// TIA Portal V17 export
// export: Created 2023-10-17T06:55:20.3967986Z, ExportSetting WithDefaults, DisplayName Totally Integrated Automation Portal, DisplayVersion V17, DisplayName TIA Portal Openness, DisplayVersion V17, DisplayName TIA Portal Version Control Interface, DisplayVersion V17, DisplayName STEP 7 Professional, DisplayVersion V17, DisplayName STEP 7 Safety, DisplayVersion V17, DisplayName WinCC Advanced, DisplayVersion V17
ORGANIZATION_BLOCK "Main"   // OB1, LAD, ProgramCycle
TITLE = "Main Program Sweep (Cycle)"
{ S7_Optimized_Access := 'TRUE' }
VERSION : 0.1
// stored: AutoNumber true, IsIECCheckEnabled false, SetENOAutomatically false
   VAR_INPUT
      Initial_Call : Bool;   // Initial call of this OB
      Remanence : Bool;   // =True, if remanent data are available
   END_VAR
   VAR_TEMP
      "Auto/Manual" : Bool;
   END_VAR
   VAR_TEMP   // added for the SCL form of the ladder/FBD networks
      _w1 : Bool;
   END_VAR
BEGIN

REGION Network 1
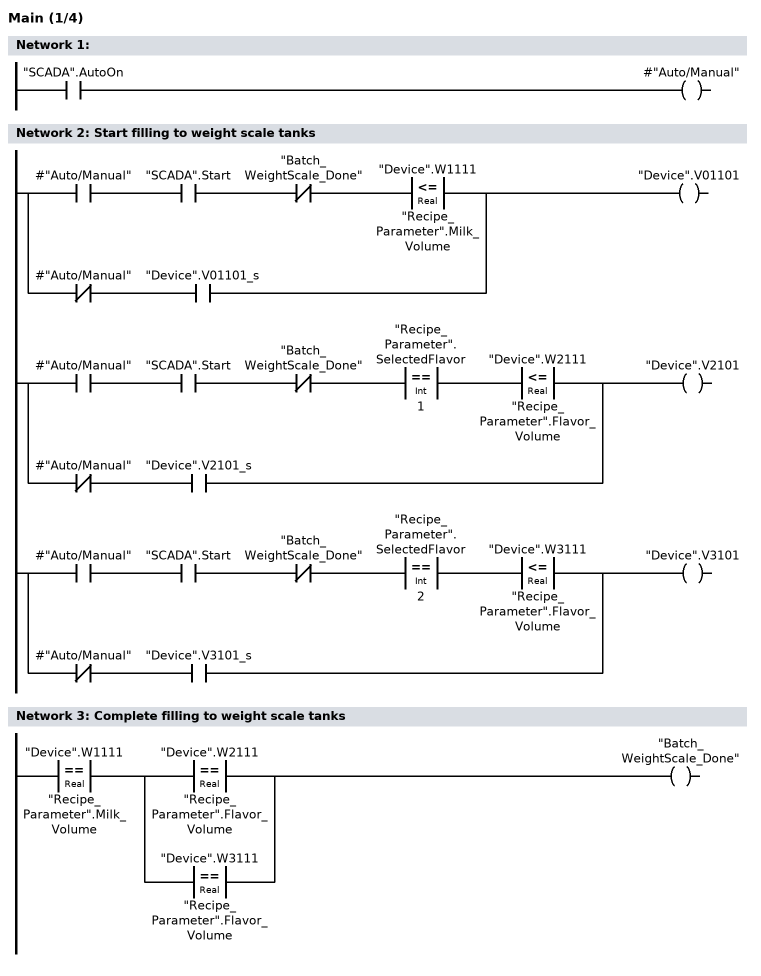
   RUNG wire#powerrail
      Contact( "SCADA".AutoOn )
      Coil( #"Auto/Manual" )
   END_RUNG
   // the same network as SCL:
   #"Auto/Manual" := "SCADA".AutoOn;
END_REGION

REGION Network 2: Start filling to weight scale tanks
   RUNG wire#powerrail
      Contact( #"Auto/Manual" )
      Contact( "SCADA".Start )
      I_Contact( "Batch_WeightScale_Done" )
      { S7_Templates := "SrcType := Real" } LE_Contact(in1 := "Device".W1111, in2 := "Recipe_Parameter".Milk_Volume)
      wire#w1
      Coil( "Device".V01101 )
   END_RUNG
   RUNG wire#powerrail
      I_Contact( #"Auto/Manual" )
      Contact( "Device".V01101_s )
   END_RUNG wire#w1
   RUNG wire#powerrail
      Contact( #"Auto/Manual" )
      Contact( "SCADA".Start )
      I_Contact( "Batch_WeightScale_Done" )
      { S7_Templates := "SrcType := Int" } EQ_Contact(in1 := "Recipe_Parameter".SelectedFlavor, in2 := 1)
      { S7_Templates := "SrcType := Real" } LE_Contact(in1 := "Device".W2111, in2 := "Recipe_Parameter".Flavor_Volume)
      wire#w2
      Coil( "Device".V2101 )
   END_RUNG
   RUNG wire#powerrail
      I_Contact( #"Auto/Manual" )
      Contact( "Device".V2101_s )
   END_RUNG wire#w2
   RUNG wire#powerrail
      Contact( #"Auto/Manual" )
      Contact( "SCADA".Start )
      I_Contact( "Batch_WeightScale_Done" )
      { S7_Templates := "SrcType := Int" } EQ_Contact(in1 := "Recipe_Parameter".SelectedFlavor, in2 := 2)
      { S7_Templates := "SrcType := Real" } LE_Contact(in1 := "Device".W3111, in2 := "Recipe_Parameter".Flavor_Volume)
      wire#w3
      Coil( "Device".V3101 )
   END_RUNG
   RUNG wire#powerrail
      I_Contact( #"Auto/Manual" )
      Contact( "Device".V3101_s )
   END_RUNG wire#w3
   // the same network as SCL:
   "Device".V01101 := (#"Auto/Manual" AND "SCADA".Start AND NOT "Batch_WeightScale_Done" AND ("Device".W1111 <= "Recipe_Parameter".Milk_Volume)) OR (NOT #"Auto/Manual" AND "Device".V01101_s);
   "Device".V2101 := (#"Auto/Manual" AND "SCADA".Start AND NOT "Batch_WeightScale_Done" AND ("Recipe_Parameter".SelectedFlavor = 1) AND ("Device".W2111 <= "Recipe_Parameter".Flavor_Volume)) OR (NOT #"Auto/Manual" AND "Device".V2101_s);
   "Device".V3101 := (#"Auto/Manual" AND "SCADA".Start AND NOT "Batch_WeightScale_Done" AND ("Recipe_Parameter".SelectedFlavor = 2) AND ("Device".W3111 <= "Recipe_Parameter".Flavor_Volume)) OR (NOT #"Auto/Manual" AND "Device".V3101_s);
END_REGION

REGION Network 3: Complete filling to weight scale tanks
   RUNG wire#powerrail
      { S7_Templates := "SrcType := Real" } EQ_Contact(in1 := "Device".W1111, in2 := "Recipe_Parameter".Milk_Volume)
      wire#w1
      { S7_Templates := "SrcType := Real" } EQ_Contact(in1 := "Device".W2111, in2 := "Recipe_Parameter".Flavor_Volume)
      wire#w2
      Coil( "Batch_WeightScale_Done" )
   END_RUNG
   RUNG wire#w1
      { S7_Templates := "SrcType := Real" } EQ_Contact(in1 := "Device".W3111, in2 := "Recipe_Parameter".Flavor_Volume)
   END_RUNG wire#w2
   // the same network as SCL:
   "Batch_WeightScale_Done" := ("Device".W1111 = "Recipe_Parameter".Milk_Volume) AND (("Device".W2111 = "Recipe_Parameter".Flavor_Volume) OR ("Device".W3111 = "Recipe_Parameter".Flavor_Volume));
END_REGION

REGION Network 4: Start filling the mixer
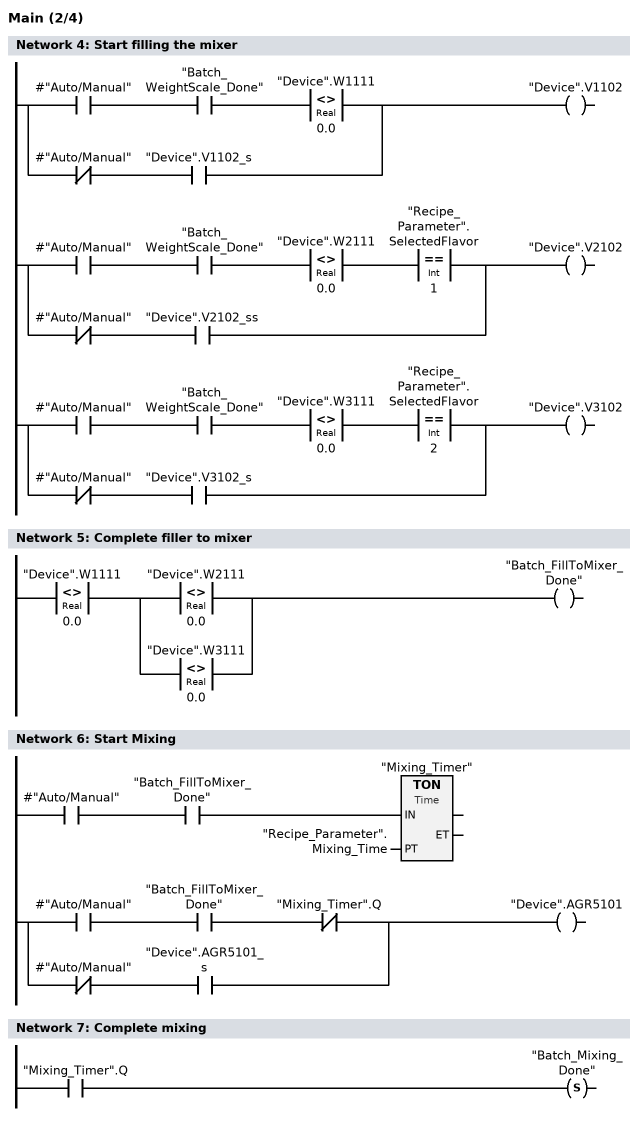
   RUNG wire#powerrail
      Contact( #"Auto/Manual" )
      Contact( "Batch_WeightScale_Done" )
      { S7_Templates := "SrcType := Real" } NE_Contact(in1 := "Device".W1111, in2 := 0.0)
      wire#w1
      Coil( "Device".V1102 )
   END_RUNG
   RUNG wire#powerrail
      I_Contact( #"Auto/Manual" )
      Contact( "Device".V1102_s )
   END_RUNG wire#w1
   RUNG wire#powerrail
      Contact( #"Auto/Manual" )
      Contact( "Batch_WeightScale_Done" )
      { S7_Templates := "SrcType := Real" } NE_Contact(in1 := "Device".W2111, in2 := 0.0)
      { S7_Templates := "SrcType := Int" } EQ_Contact(in1 := "Recipe_Parameter".SelectedFlavor, in2 := 1)
      wire#w2
      Coil( "Device".V2102 )
   END_RUNG
   RUNG wire#powerrail
      I_Contact( #"Auto/Manual" )
      Contact( "Device".V2102_ss )
   END_RUNG wire#w2
   RUNG wire#powerrail
      Contact( #"Auto/Manual" )
      Contact( "Batch_WeightScale_Done" )
      { S7_Templates := "SrcType := Real" } NE_Contact(in1 := "Device".W3111, in2 := 0.0)
      { S7_Templates := "SrcType := Int" } EQ_Contact(in1 := "Recipe_Parameter".SelectedFlavor, in2 := 2)
      wire#w3
      Coil( "Device".V3102 )
   END_RUNG
   RUNG wire#powerrail
      I_Contact( #"Auto/Manual" )
      Contact( "Device".V3102_s )
   END_RUNG wire#w3
   // the same network as SCL:
   "Device".V1102 := (#"Auto/Manual" AND "Batch_WeightScale_Done" AND ("Device".W1111 <> 0.0)) OR (NOT #"Auto/Manual" AND "Device".V1102_s);
   "Device".V2102 := (#"Auto/Manual" AND "Batch_WeightScale_Done" AND ("Device".W2111 <> 0.0) AND ("Recipe_Parameter".SelectedFlavor = 1)) OR (NOT #"Auto/Manual" AND "Device".V2102_ss);
   "Device".V3102 := (#"Auto/Manual" AND "Batch_WeightScale_Done" AND ("Device".W3111 <> 0.0) AND ("Recipe_Parameter".SelectedFlavor = 2)) OR (NOT #"Auto/Manual" AND "Device".V3102_s);
END_REGION

REGION Network 5: Complete filler to mixer
   RUNG wire#powerrail
      { S7_Templates := "SrcType := Real" } NE_Contact(in1 := "Device".W1111, in2 := 0.0)
      wire#w1
      { S7_Templates := "SrcType := Real" } NE_Contact(in1 := "Device".W2111, in2 := 0.0)
      wire#w2
      Coil( "Batch_FillToMixer_Done" )
   END_RUNG
   RUNG wire#w1
      { S7_Templates := "SrcType := Real" } NE_Contact(in1 := "Device".W3111, in2 := 0.0)
   END_RUNG wire#w2
   // the same network as SCL:
   "Batch_FillToMixer_Done" := ("Device".W1111 <> 0.0) AND (("Device".W2111 <> 0.0) OR ("Device".W3111 <> 0.0));
END_REGION

REGION Network 6: Start Mixing
   RUNG wire#powerrail
      Contact( #"Auto/Manual" )
      Contact( "Batch_FillToMixer_Done" )
      { S7_Templates := "time_type := Time" } "Mixing_Timer".TON(pt := "Recipe_Parameter".Mixing_Time, et =>)
   END_RUNG
   RUNG wire#powerrail
      Contact( #"Auto/Manual" )
      Contact( "Batch_FillToMixer_Done" )
      I_Contact( "Mixing_Timer".Q )
      wire#w1
      Coil( "Device".AGR5101 )
   END_RUNG
   RUNG wire#powerrail
      I_Contact( #"Auto/Manual" )
      Contact( "Device".AGR5101_s )
   END_RUNG wire#w1
   // the same network as SCL:
   "Mixing_Timer".TON(IN := #"Auto/Manual" AND "Batch_FillToMixer_Done", PT := "Recipe_Parameter".Mixing_Time);
   "Device".AGR5101 := (#"Auto/Manual" AND "Batch_FillToMixer_Done" AND NOT "Mixing_Timer".Q) OR (NOT #"Auto/Manual" AND "Device".AGR5101_s);
END_REGION

REGION Network 7: Complete mixing
   RUNG wire#powerrail
      Contact( "Mixing_Timer".Q )
      S_Coil( "Batch_Mixing_Done" )
   END_RUNG
   // the same network as SCL:
   IF "Mixing_Timer".Q THEN "Batch_Mixing_Done" := TRUE; END_IF;
END_REGION

REGION Network 8: Start filling to pasteurising machine
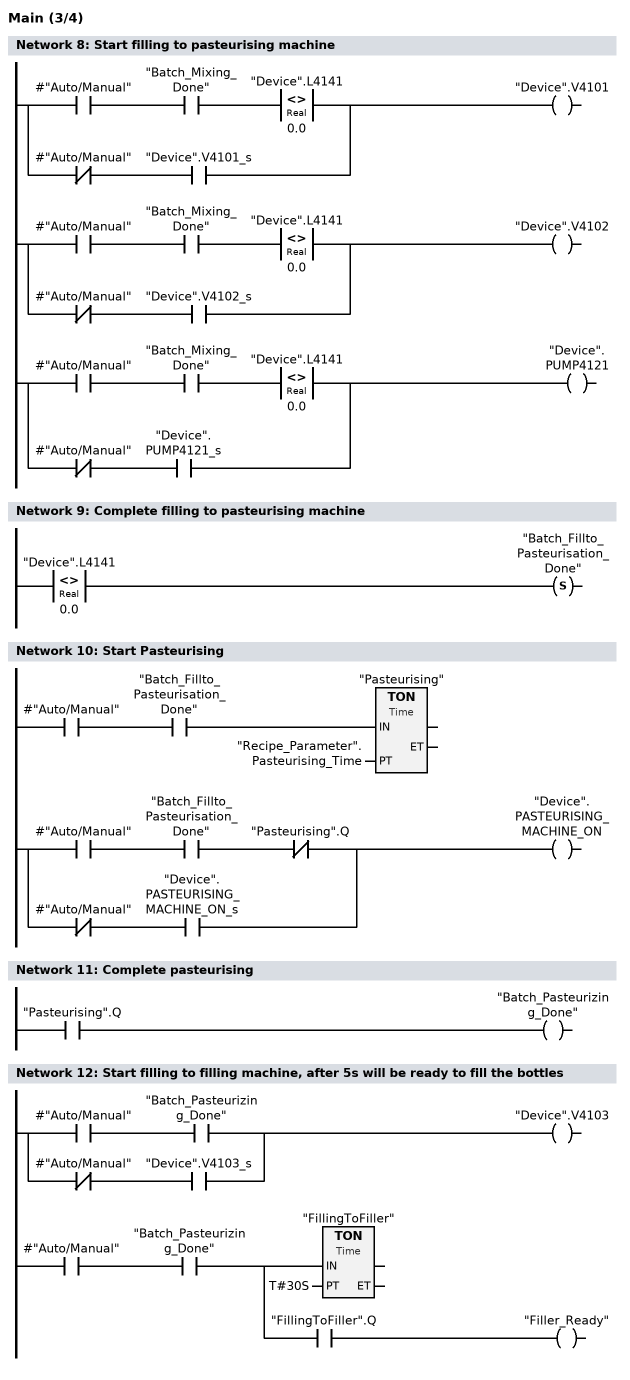
   RUNG wire#powerrail
      Contact( #"Auto/Manual" )
      Contact( "Batch_Mixing_Done" )
      { S7_Templates := "SrcType := Real" } NE_Contact(in1 := "Device".L4141, in2 := 0.0)
      wire#w1
      Coil( "Device".V4101 )
   END_RUNG
   RUNG wire#powerrail
      I_Contact( #"Auto/Manual" )
      Contact( "Device".V4101_s )
   END_RUNG wire#w1
   RUNG wire#powerrail
      Contact( #"Auto/Manual" )
      Contact( "Batch_Mixing_Done" )
      { S7_Templates := "SrcType := Real" } NE_Contact(in1 := "Device".L4141, in2 := 0.0)
      wire#w2
      Coil( "Device".V4102 )
   END_RUNG
   RUNG wire#powerrail
      I_Contact( #"Auto/Manual" )
      Contact( "Device".V4102_s )
   END_RUNG wire#w2
   RUNG wire#powerrail
      Contact( #"Auto/Manual" )
      Contact( "Batch_Mixing_Done" )
      { S7_Templates := "SrcType := Real" } NE_Contact(in1 := "Device".L4141, in2 := 0.0)
      wire#w3
      Coil( "Device".PUMP4121 )
   END_RUNG
   RUNG wire#powerrail
      I_Contact( #"Auto/Manual" )
      Contact( "Device".PUMP4121_s )
   END_RUNG wire#w3
   // the same network as SCL:
   "Device".V4101 := (#"Auto/Manual" AND "Batch_Mixing_Done" AND ("Device".L4141 <> 0.0)) OR (NOT #"Auto/Manual" AND "Device".V4101_s);
   "Device".V4102 := (#"Auto/Manual" AND "Batch_Mixing_Done" AND ("Device".L4141 <> 0.0)) OR (NOT #"Auto/Manual" AND "Device".V4102_s);
   "Device".PUMP4121 := (#"Auto/Manual" AND "Batch_Mixing_Done" AND ("Device".L4141 <> 0.0)) OR (NOT #"Auto/Manual" AND "Device".PUMP4121_s);
END_REGION

REGION Network 9: Complete filling to pasteurising machine
   RUNG wire#powerrail
      { S7_Templates := "SrcType := Real" } NE_Contact(in1 := "Device".L4141, in2 := 0.0)
      S_Coil( "Batch_Fillto_Pasteurisation_Done" )
   END_RUNG
   // the same network as SCL:
   IF "Device".L4141 <> 0.0 THEN "Batch_Fillto_Pasteurisation_Done" := TRUE; END_IF;
END_REGION

REGION Network 10: Start Pasteurising
   RUNG wire#powerrail
      Contact( #"Auto/Manual" )
      Contact( "Batch_Fillto_Pasteurisation_Done" )
      { S7_Templates := "time_type := Time" } "Pasteurising".TON(pt := "Recipe_Parameter".Pasteurising_Time, et =>)
   END_RUNG
   RUNG wire#powerrail
      Contact( #"Auto/Manual" )
      Contact( "Batch_Fillto_Pasteurisation_Done" )
      I_Contact( "Pasteurising".Q )
      wire#w1
      Coil( "Device".PASTEURISING_MACHINE_ON )
   END_RUNG
   RUNG wire#powerrail
      I_Contact( #"Auto/Manual" )
      Contact( "Device".PASTEURISING_MACHINE_ON_s )
   END_RUNG wire#w1
   // the same network as SCL:
   "Pasteurising".TON(IN := #"Auto/Manual" AND "Batch_Fillto_Pasteurisation_Done",
                      PT := "Recipe_Parameter".Pasteurising_Time);
   "Device".PASTEURISING_MACHINE_ON := (#"Auto/Manual" AND "Batch_Fillto_Pasteurisation_Done" AND NOT "Pasteurising".Q) OR (NOT #"Auto/Manual" AND "Device".PASTEURISING_MACHINE_ON_s);
END_REGION

REGION Network 11: Complete pasteurising
   RUNG wire#powerrail
      Contact( "Pasteurising".Q )
      Coil( "Batch_Pasteurizing_Done" )
   END_RUNG
   // the same network as SCL:
   "Batch_Pasteurizing_Done" := "Pasteurising".Q;
END_REGION

REGION Network 12: Start filling to filling machine, after 5s will be ready to fill the bottles
   RUNG wire#powerrail
      Contact( #"Auto/Manual" )
      Contact( "Batch_Pasteurizing_Done" )
      wire#w1
      Coil( "Device".V4103 )
   END_RUNG
   RUNG wire#powerrail
      I_Contact( #"Auto/Manual" )
      Contact( "Device".V4103_s )
   END_RUNG wire#w1
   RUNG wire#powerrail
      Contact( #"Auto/Manual" )
      Contact( "Batch_Pasteurizing_Done" )
      wire#w2
      { S7_Templates := "time_type := Time" } "FillingToFiller".TON(pt := T#30S, et =>)
   END_RUNG
   RUNG wire#w2
      Contact( "FillingToFiller".Q )
      Coil( "Filler_Ready" )
   END_RUNG
   // the same network as SCL:
   "Device".V4103 := (#"Auto/Manual" AND "Batch_Pasteurizing_Done") OR (NOT #"Auto/Manual" AND "Device".V4103_s);
   #_w1 := #"Auto/Manual" AND "Batch_Pasteurizing_Done";
   "FillingToFiller".TON(IN := #_w1, PT := T#30S);
   "Filler_Ready" := #_w1 AND "FillingToFiller".Q;
END_REGION

REGION Network 13: Run filler until level of feed until 0.5 liters
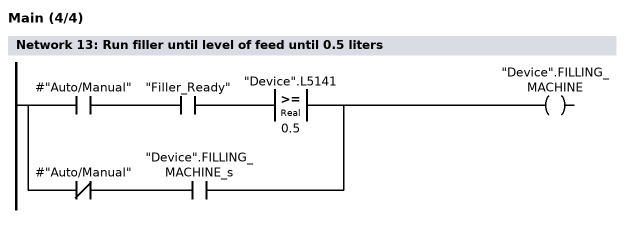
   RUNG wire#powerrail
      Contact( #"Auto/Manual" )
      Contact( "Filler_Ready" )
      { S7_Templates := "SrcType := Real" } GE_Contact(in1 := "Device".L5141, in2 := 0.5)
      wire#w1
      Coil( "Device".FILLING_MACHINE )
   END_RUNG
   RUNG wire#powerrail
      I_Contact( #"Auto/Manual" )
      Contact( "Device".FILLING_MACHINE_s )
   END_RUNG wire#w1
   // the same network as SCL:
   "Device".FILLING_MACHINE := (#"Auto/Manual" AND "Filler_Ready" AND ("Device".L5141 >= 0.5)) OR (NOT #"Auto/Manual" AND "Device".FILLING_MACHINE_s);
END_REGION
END_ORGANIZATION_BLOCK
